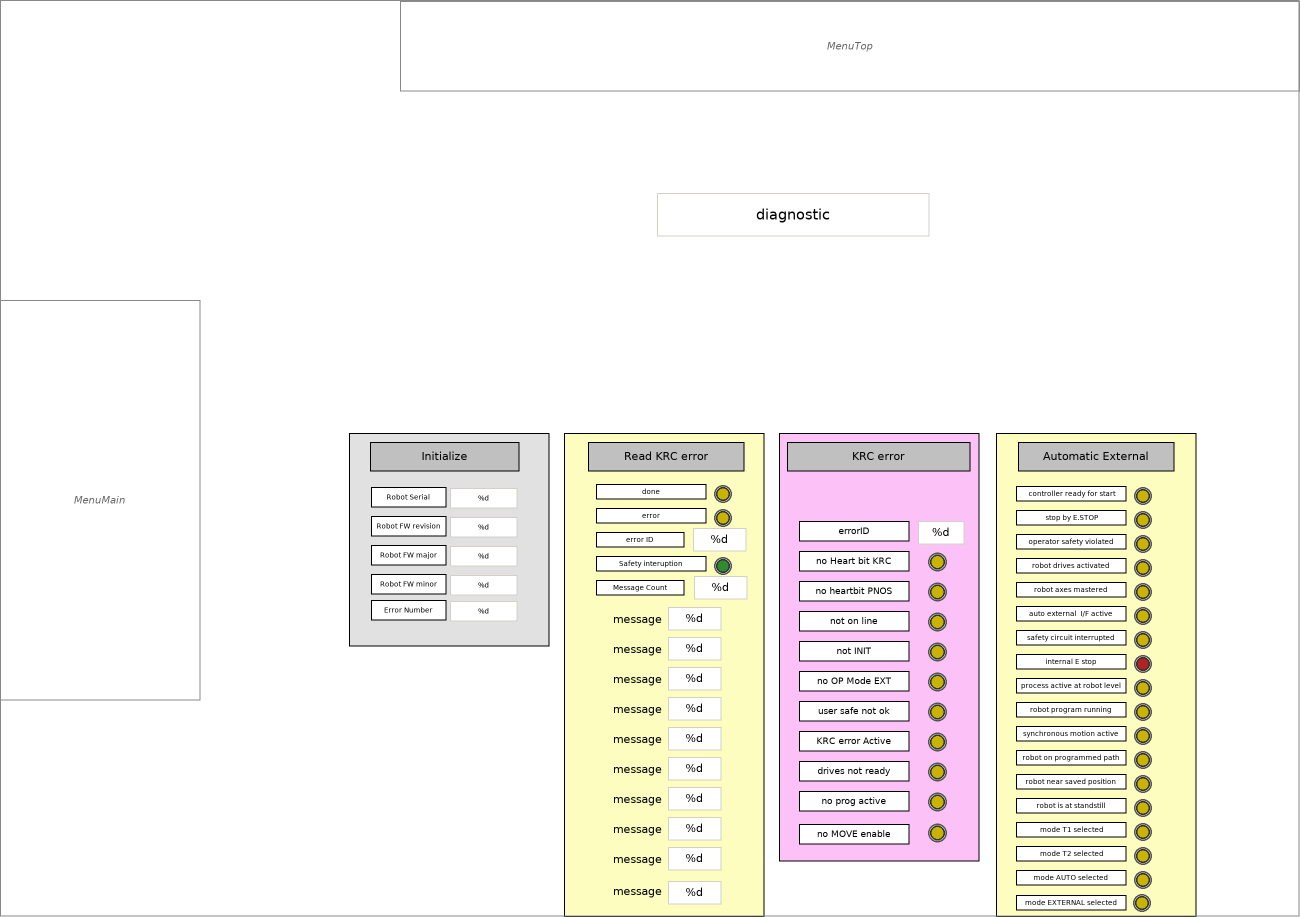
VISUALIZATION diagnostic  // 1300x917
    Rectangle (996,433 200x484), text variable: MAIN.fbKRC_Error.ErrorID
    Rectangle (349,433 200x213)
    Rectangle (779,433 200x428)
    Frame (400,1 900x90)
        shows MenuTop()
    Frame (0,300 200x400)
        shows MenuMain()
    Textfield (657,193 272x43), "diagnostic"
    Lamp1 (1123,486 40x20), variable: MAIN.fbKRC_AutomaticExternal.RC_RDY1, style: Lamp-Lamp1-Yellow
    Lamp1 (1123,510 40x20), variable: MAIN.fbKRC_AutomaticExternal.ALARM_STOP, style: Lamp-Lamp1-Yellow
    Lamp1 (1123,534 40x20), variable: MAIN.fbKRC_AutomaticExternal.USER_SAFE, style: Lamp-Lamp1-Yellow
    Lamp1 (1123,558 40x20), variable: MAIN.fbKRC_AutomaticExternal.PERI_RDY, style: Lamp-Lamp1-Yellow
    Lamp1 (1123,582 40x20), variable: MAIN.fbKRC_AutomaticExternal.ROB_CAL, style: Lamp-Lamp1-Yellow
    Lamp1 (1123,606 40x20), variable: MAIN.fbKRC_AutomaticExternal.IO_ACTCONF, style: Lamp-Lamp1-Yellow
    Rectangle (371,516 75x20), "Robot FW revision"
    Rectangle (371,545 75x20), "Robot FW major"
    Rectangle (371,574 75x20), "Robot FW minor"
    Textfield (450,517 67x20), "%d", text variable: MAIN.fbKRC_Initialize.KRC_Revision
    Textfield (450,546 67x20), "%d", text variable: MAIN.fbKRC_Initialize.KRC_Major
    Textfield (450,575 67x20), "%d", text variable: MAIN.fbKRC_Initialize.KRC_Minor
    Rectangle (371,487 75x20), "Robot Serial"
    Textfield (450,488 67x20), "%d", text variable: MAIN.fbKRC_Initialize.KRC_Serial
    Rectangle (1018,442 156x29), "Automatic External", text variable: GVL.HMI_Error_General_ID, colour toggle: GVL.HMI_Error_General
    Rectangle (1016,486 110x15), "controller ready for start", text variable: GVL.HMI_Error_General_ID, colour toggle: GVL.HMI_Error_General
    Rectangle (1016,510 110x15), "stop by E.STOP", text variable: GVL.HMI_Error_General_ID, colour toggle: GVL.HMI_Error_General
    Rectangle (1016,534 110x15), "operator safety violated", text variable: GVL.HMI_Error_General_ID, colour toggle: GVL.HMI_Error_General
    Rectangle (1016,558 110x15), "robot drives activated", text variable: GVL.HMI_Error_General_ID, colour toggle: GVL.HMI_Error_General
    Rectangle (1016,582 110x15), "robot axes mastered", text variable: GVL.HMI_Error_General_ID, colour toggle: GVL.HMI_Error_General
    Rectangle (1016,606 110x15), "auto external I/F active", text variable: GVL.HMI_Error_General_ID, colour toggle: GVL.HMI_Error_General
    Lamp1 (1123,630 40x20), variable: MAIN.fbKRC_AutomaticExternal.STOPMESS, style: Lamp-Lamp1-Yellow
    Lamp1 (1123,654 40x20), variable: MAIN.NOT_INT_E_STOP, style: Lamp-Lamp1-Red
    Lamp1 (1123,678 40x20), variable: MAIN.fbKRC_AutomaticExternal.PRO_ACT, style: Lamp-Lamp1-Yellow
    Rectangle (1016,630 110x15), "safety circuit interrupted", text variable: GVL.HMI_Error_General_ID, colour toggle: GVL.HMI_Error_General
    Rectangle (1016,654 110x15), "internal E stop", text variable: GVL.HMI_Error_General_ID, colour toggle: GVL.HMI_Error_General
    Rectangle (1016,678 110x15), "process active at robot level", text variable: GVL.HMI_Error_General_ID, colour toggle: GVL.HMI_Error_General
    Lamp1 (1123,702 40x20), variable: MAIN.fbKRC_AutomaticExternal.APPL_RUN, style: Lamp-Lamp1-Yellow
    Rectangle (1016,702 110x15), "robot program running", text variable: GVL.HMI_Error_General_ID, colour toggle: GVL.HMI_Error_General
    Lamp1 (1123,726 40x20), variable: MAIN.fbKRC_AutomaticExternal.PRO_MOVE, style: Lamp-Lamp1-Yellow
    Lamp1 (1123,750 40x20), variable: MAIN.fbKRC_AutomaticExternal.ON_PATH, style: Lamp-Lamp1-Yellow
    Lamp1 (1123,774 40x20), variable: MAIN.fbKRC_AutomaticExternal.NEAR_POSRET, style: Lamp-Lamp1-Yellow
    Rectangle (1016,726 110x15), "synchronous motion active", text variable: GVL.HMI_Error_General_ID, colour toggle: GVL.HMI_Error_General
    Rectangle (1016,750 110x15), "robot on programmed path", text variable: GVL.HMI_Error_General_ID, colour toggle: GVL.HMI_Error_General
    Rectangle (1016,774 110x15), "robot near saved position", text variable: GVL.HMI_Error_General_ID, colour toggle: GVL.HMI_Error_General
    Rectangle (1016,798 110x15), "robot is at standstill", text variable: GVL.HMI_Error_General_ID, colour toggle: GVL.HMI_Error_General
    Rectangle (1016,822 110x15), "mode T1 selected", text variable: GVL.HMI_Error_General_ID, colour toggle: GVL.HMI_Error_General
    Rectangle (1016,846 110x15), "mode T2 selected", text variable: GVL.HMI_Error_General_ID, colour toggle: GVL.HMI_Error_General
    Rectangle (1016,870 110x15), "mode AUTO selected", text variable: GVL.HMI_Error_General_ID, colour toggle: GVL.HMI_Error_General
    Rectangle (1016,895 110x15), "mode EXTERNAL selected", text variable: GVL.HMI_Error_General_ID, colour toggle: GVL.HMI_Error_General
    Lamp1 (1123,798 40x20), variable: MAIN.fbKRC_AutomaticExternal.PRO_ACT, style: Lamp-Lamp1-Yellow
    Lamp1 (1123,822 40x20), variable: MAIN.fbKRC_AutomaticExternal.T1, style: Lamp-Lamp1-Yellow
    Lamp1 (1123,846 40x20), variable: MAIN.fbKRC_AutomaticExternal.T2, style: Lamp-Lamp1-Yellow
    Lamp1 (1123,870 40x20), variable: MAIN.fbKRC_AutomaticExternal.AUT, style: Lamp-Lamp1-Yellow
    Lamp1 (1123,893 38x20), variable: MAIN.fbKRC_AutomaticExternal.EXT, style: Lamp-Lamp1-Yellow
    Rectangle (370,442 149x29), "Initialize", text variable: GVL.HMI_Error_General_ID, colour toggle: GVL.HMI_Error_General
    Rectangle (371,600 75x20), "Error Number"
    Textfield (450,601 67x20), "%d", text variable: MAIN.fbKRC_Initialize.Error
    Rectangle (787,442 183x29), "KRC error", text variable: GVL.HMI_Error_General_ID, colour toggle: GVL.HMI_Error_General
    Rectangle (799,521 110x20), "errorID"
    Rectangle (799,551 110x20), "no Heart bit KRC"
    Rectangle (799,581 110x20), "no heartbit PNOS"
    Rectangle (799,611 110x20), "not on line"
    Rectangle (799,641 110x20), "not INIT"
    Rectangle (799,671 110x20), "no OP Mode EXT"
    Rectangle (799,701 110x20), "user safe not ok"
    Rectangle (799,731 110x20), "KRC error Active"
    Rectangle (799,761 110x20), "drives not ready"
    Rectangle (799,791 110x20), "no prog active"
    Rectangle (799,824 110x20), "no MOVE enable"
    Lamp1 (926,551 23x22), variable: MAIN.fbKRC_Error.NoHeartbeatKRC, style: Lamp-Lamp1-Yellow
    Lamp1 (926,581 23x22), variable: MAIN.fbKRC_Error.NoHeartbeatPCOS, style: Lamp-Lamp1-Yellow
    Lamp1 (926,611 23x22), variable: MAIN.fbKRC_Error.NoMoveEnable, style: Lamp-Lamp1-Yellow
    Lamp1 (926,641 23x22), variable: MAIN.fbKRC_Error.NotInitialized, style: Lamp-Lamp1-Yellow
    Lamp1 (926,671 23x22), variable: MAIN.fbKRC_Error.NoOpModeExt, style: Lamp-Lamp1-Yellow
    Lamp1 (926,701 23x22), variable: MAIN.fbKRC_Error.UserSafeNotOK, style: Lamp-Lamp1-Yellow
    Lamp1 (926,731 23x22), variable: MAIN.fbKRC_Error.KrcErrorActive, style: Lamp-Lamp1-Yellow
    Lamp1 (926,761 23x22), variable: MAIN.fbKRC_Error.DrivesNotReady, style: Lamp-Lamp1-Yellow
    Lamp1 (926,791 23x22), variable: MAIN.fbKRC_Error.NoProgActive, style: Lamp-Lamp1-Yellow
    Lamp1 (926,822 23x22), variable: MAIN.fbKRC_Error.NoMoveEnable, style: Lamp-Lamp1-Yellow
    Textfield (918,521 46x23), "%d", text variable: MAIN.fbKRC_Error.ErrorID
    Rectangle (564,433 200x484), text variable: MAIN.fbKRC_Error.ErrorID
    Lamp1 (703,484 40x20), variable: MAIN.ReadKRCError.Done, style: Lamp-Lamp1-Yellow
    Lamp1 (703,508 40x20), variable: MAIN.ReadKRCError.Error, style: Lamp-Lamp1-Yellow
    Lamp1 (703,556 40x20), variable: NOT(MAIN.ReadKRCError.STOPMESS), style: Lamp-Lamp1-Green
    Rectangle (588,442 156x29), "Read KRC error", text variable: GVL.HMI_Error_General_ID, colour toggle: GVL.HMI_Error_General
    Rectangle (596,484 110x15), "done", text variable: GVL.HMI_Error_General_ID, colour toggle: GVL.HMI_Error_General
    Rectangle (596,508 110x15), "error", text variable: GVL.HMI_Error_General_ID, colour toggle: GVL.HMI_Error_General
    Rectangle (596,532 88x15), "error ID", text variable: GVL.HMI_Error_General_ID, colour toggle: GVL.HMI_Error_General
    Rectangle (596,556 110x15), "Safety interuption", text variable: MAIN.ReadKRCError.STOPMESS, colour toggle: GVL.HMI_Error_General
    Rectangle (596,580 88x15), "Message Count", text variable: GVL.HMI_Error_General_ID, colour toggle: GVL.HMI_Error_General
    Textfield (693,528 53x23), "%d", text variable: MAIN.ReadKRCError.ErrorID
    Textfield (694,576 53x23), "%d", text variable: MAIN.ReadKRCError.ErrorID
    Textfield (668,607 53x23), "%d", text variable: MAIN.ReadKRCError.Message1
    Textfield (668,637 53x23), "%d", text variable: MAIN.ReadKRCError.Message2
    Textfield (668,667 53x23), "%d", text variable: MAIN.ReadKRCError.Message3
    Textfield (668,697 53x23), "%d", text variable: MAIN.ReadKRCError.Message4
    Textfield (668,727 53x23), "%d", text variable: MAIN.ReadKRCError.Message5
    Textfield (668,757 53x23), "%d", text variable: MAIN.ReadKRCError.Message6
    Textfield (668,787 53x23), "%d", text variable: MAIN.ReadKRCError.Message7
    Textfield (668,817 53x23), "%d", text variable: MAIN.ReadKRCError.Message8
    Textfield (668,847 53x23), "%d", text variable: MAIN.ReadKRCError.Message9
    Textfield (668,881 53x23), "%d", text variable: MAIN.ReadKRCError.Message10
    Label (612,605 51x29), "message"
    Label (612,635 51x29), "message"
    Label (612,665 51x29), "message"
    Label (612,695 51x29), "message"
    Label (612,725 51x29), "message"
    Label (612,755 51x29), "message"
    Label (612,785 51x29), "message"
    Label (612,815 51x29), "message"
    Label (612,845 51x29), "message"
    Label (612,877 51x29), "message"
END_VISUALIZATION

(* stored: Version 1.1.0.1, ProductVersion 3.1.4024.10
   Visu diagnostic: Id {3a88a4dd-0fd6-4b4d-bce8-1870d92c29bc} *)
